// TIA Portal V17 program export: 0 tag tables, 0 data types, 0 data blocks, 2 code blocks (in call order from the OBs), 0 instance data blocks

ORGANIZATION_BLOCK "Main"   // OB1, LAD, ProgramCycle
TITLE = "Main Program Sweep (Cycle)"
{ S7_Optimized_Access := 'TRUE' }
VERSION : 0.1
// stored: AutoNumber true, IsIECCheckEnabled false, SetENOAutomatically false
   VAR_INPUT
      Initial_Call : Bool;   // Initial call of this OB
      Remanence : Bool;   // =True, if remanent data are available
   END_VAR
   VAR_TEMP
      temperature : Real;
   END_VAR
   VAR CONSTANT
      temperatureMin : Real := 0.0;
      temperatureMax : Real := 100.0;
   END_VAR
BEGIN

REGION Network 1: Scale analog input temperature on IW64
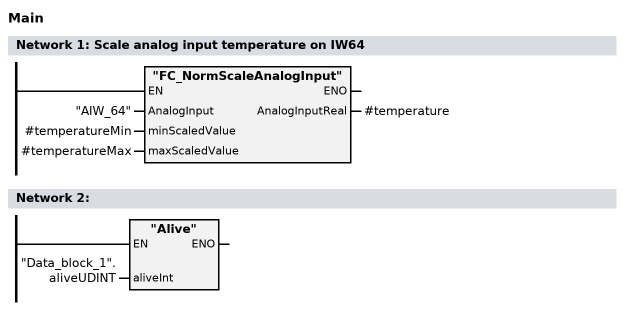
   RUNG wire#powerrail
      "FC_NormScaleAnalogInput"(AnalogInput := "AIW_64", minScaledValue := #temperatureMin, maxScaledValue := #temperatureMax, AnalogInputReal => #temperature)
   END_RUNG
   // the same network as SCL:
   "FC_NormScaleAnalogInput"(AnalogInput := "AIW_64",
                           minScaledValue := #temperatureMin,
                           maxScaledValue := #temperatureMax,
                           AnalogInputReal => #temperature);
END_REGION

REGION Network 2
   RUNG wire#powerrail
      "Alive"(aliveInt := "Data_block_1".aliveUDINT)
   END_RUNG
   // the same network as SCL:
   "Alive"(aliveInt := "Data_block_1".aliveUDINT);
END_REGION
END_ORGANIZATION_BLOCK

FUNCTION "FC_NormScaleAnalogInput" : Void   // FC1, LAD
{ S7_Optimized_Access := 'TRUE' }
VERSION : 0.1
// stored: AutoNumber true, IsIECCheckEnabled false, SetENOAutomatically false, UDAEnableTagReadback false
   VAR_INPUT
      AnalogInput : Int;   // Analog input [value 0 - 27648]
      minScaledValue : Real;   // lower value for scaled value Real
      maxScaledValue : Real;   // Upper value for scaled value Real
   END_VAR
   VAR_OUTPUT
      AnalogInputReal : Real;   // Scaled analog value Real
   END_VAR
   VAR_TEMP
      normAnalogValue : Real;
   END_VAR
   VAR CONSTANT
      LOWERINT : Int := 0;
      UPPERINT : Int := 27648;
   END_VAR
BEGIN

REGION Network 1
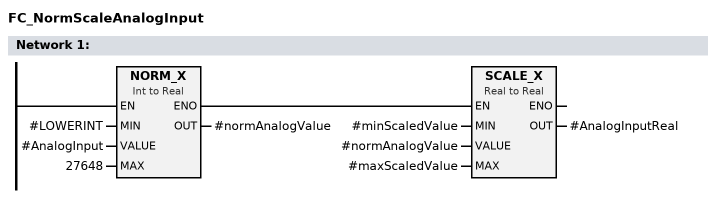
   RUNG wire#powerrail
      { S7_Templates := "[SrcType := Int, DestType := Real]" } Normalize(min := #LOWERINT, value := #AnalogInput, max := 27648, out => #normAnalogValue)
      { S7_Templates := "[SrcType := Real, DestType := Real]" } Scale(min := #minScaledValue, value := #normAnalogValue, max := #maxScaledValue, out => #AnalogInputReal)
   END_RUNG
   // the same network as SCL:
   #normAnalogValue := NORM_X(MIN := #LOWERINT, VALUE := #AnalogInput, MAX := 27648);
   #AnalogInputReal := SCALE_X(MIN := #minScaledValue, VALUE := #normAnalogValue, MAX := #maxScaledValue);
END_REGION
END_FUNCTION
